FUNCTION_BLOCK fb_gm_removeLens
VAR_INPUT
	in_flg_run: BOOL;
END_VAR
VAR_OUTPUT
	out_flg_Done: BOOL;
END_VAR
VAR
	SFCInit: BOOL;
	trn_checkVacDone: BOOL;
	trn_rmoveLensThetaDone: BOOL;
	var_process: INT;
	trn_removeLensDone: BOOL;
	trn_removeLen_stocker_eject_Done : BOOL;
	trn_removeLen_stocker_fiber_Done : BOOL;
	trn_removeLen_measurement_eject_Done : BOOL;
	trn_removeLen_measurement_fiber_Done : BOOL;
	timer: TON;
	timer2: TON;
END_VAR

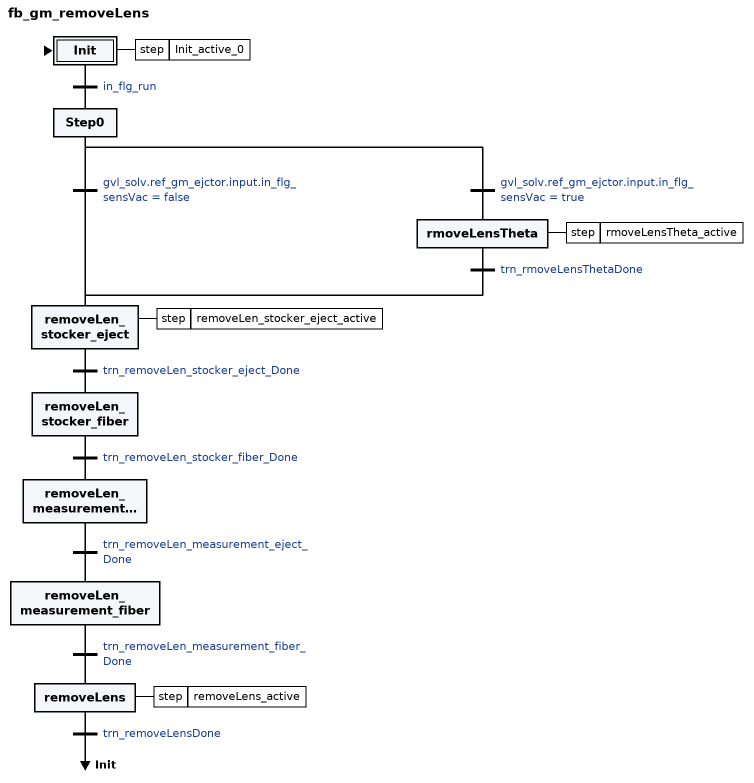
INITIAL_STEP Init:
    Init_active_0(N);  // step action
END_STEP
TRANSITION FROM Init TO Step0
    := in_flg_run;
END_TRANSITION
STEP Step0:
END_STEP
TRANSITION FROM Step0 TO removeLen_stocker_eject
    := gvl_solv.ref_gm_ejctor.input.in_flg_sensVac = false;
END_TRANSITION
TRANSITION FROM Step0 TO rmoveLensTheta
    := gvl_solv.ref_gm_ejctor.input.in_flg_sensVac = true;
END_TRANSITION
STEP rmoveLensTheta:
    rmoveLensTheta_active(N);  // step action
END_STEP
TRANSITION FROM rmoveLensTheta TO removeLen_stocker_eject
    := trn_rmoveLensThetaDone;
END_TRANSITION
STEP removeLen_stocker_eject:
    removeLen_stocker_eject_active(N);  // step action
END_STEP
TRANSITION FROM removeLen_stocker_eject TO removeLen_stocker_fiber
    := trn_removeLen_stocker_eject_Done;
END_TRANSITION
STEP removeLen_stocker_fiber:
END_STEP
TRANSITION FROM removeLen_stocker_fiber TO removeLen_measurement_eject
    := trn_removeLen_stocker_fiber_Done;
END_TRANSITION
STEP removeLen_measurement_eject:
END_STEP
TRANSITION FROM removeLen_measurement_eject TO removeLen_measurement_fiber
    := trn_removeLen_measurement_eject_Done;
END_TRANSITION
STEP removeLen_measurement_fiber:
END_STEP
TRANSITION FROM removeLen_measurement_fiber TO removeLens
    := trn_removeLen_measurement_fiber_Done;
END_TRANSITION
STEP removeLens:
    removeLens_active(N);  // step action
END_STEP
TRANSITION FROM removeLens TO Init
    := trn_removeLensDone;
END_TRANSITION

ACTION Init_active:
trn_removeLensDOne := false;
END_ACTION

ACTION Init_active_0:
out_flg_done := false;
END_ACTION

PROPERTY p_Init : BOOL
GET
p_Init := THIS^.SFCInit;
END_GET
SET
THIS^.SFCInit := p_Init;
END_SET
END_PROPERTY

ACTION removeLen_stocker_eject_active:
IF removeLen_stocker_eject._x AND removeLen_stocker_eject.x = FALSE THEN
	trn_removeLensDone := FALSE;
	timer.IN := FALSE;
	timer2.IN := FALSE;
	gvl_elecylinder.fbi_gm_axisPickUp.in_flg_run := FALSE;
	gvl_elecylinder.fbi_gm_axisPickUp.in_var_moveMode := eP_eleMoveMode.eleB;
	gvl_solv.fbi_gm_ejector.in_flg_run := FALSE;
	gvl_solv.fbi_gm_ejector.in_var_vacMode := eP_ejeVacMode.halt;
	gvl_axis.ref_r.Execute := FALSE;
	gvl_solv.fbi_gm_chuck.in_var_moveMode := eP_svMoveMode.svB;
	gvl_solv.fbi_gm_chuck.in_flg_run := FALSE;
	gvl_solv.fbi_gm_push.in_var_moveMode := eP_svMoveMode.svB;
	gvl_solv.fbi_gm_push.in_flg_run := FALSE;
	gvl_axis.ref_r.Position := gvl_param.var_productInfo[gvl_param.var_currentProductID].teachPos.gm_rotary.pickUp;
	var_process := 0;
ELSIF removeLen_stocker_eject._x AND removeLen_stocker_eject.x THEN
	CASE var_process OF
		0:
			IF gvl_io.flg_gm_fiberSens THEN
				var_process := 1;
			ELSE
				var_process := 100;
			END_IF
		1:
			
			
		
		
		100:
			trn_removeLensDone := TRUE;

	END_CASE
END_IF
END_ACTION

ACTION removeLens_active:
IF removeLens._x AND removeLens.x = FALSE THEN
	trn_removeLensDone := FALSE;
	timer.IN := FALSE;
	timer2.IN := FALSE;
	gvl_elecylinder.fbi_gm_axisPickUp.in_flg_run := FALSE;
	gvl_elecylinder.fbi_gm_axisPickUp.in_var_moveMode := eP_eleMoveMode.eleB;
	gvl_solv.fbi_gm_ejector.in_flg_run := FALSE;
	gvl_solv.fbi_gm_ejector.in_var_vacMode := eP_ejeVacMode.halt;
	gvl_axis.ref_r.Execute := FALSE;
	gvl_solv.fbi_gm_chuck.in_var_moveMode := eP_svMoveMode.svB;
	gvl_solv.fbi_gm_chuck.in_flg_run := FALSE;
	gvl_solv.fbi_gm_push.in_var_moveMode := eP_svMoveMode.svB;
	gvl_solv.fbi_gm_push.in_flg_run := FALSE;
	gvl_axis.ref_r.Position := gvl_param.var_productInfo[gvl_param.var_currentProductID].teachPos.gm_rotary.pickUp;
	var_process := 0;
ELSIF removeLens._x AND removeLens.x THEN
	CASE var_process OF
		0:
			IF gvl_io.flg_gm_fiberSens THEN
				//gvl_solv.fbi_gm_chuck.in_flg_run := TRUE;
				gvl_solv.fbi_gm_ejector.in_var_vacMode := eP_ejeVacMode.break;
				gvl_solv.fbi_gm_ejector.in_flg_run := TRUE;
				var_process := 15;
			ELSE
				gvl_solv.fbi_gm_ejector.in_var_vacMode := eP_ejeVacMode.break;
				gvl_solv.fbi_gm_ejector.in_flg_run := TRUE;
				var_process := 15;
			END_IF
		1:
			IF gvl_solv.fbi_gm_chuck.out_flg_Done THEN
				gvl_solv.fbi_gm_chuck.in_var_moveMode := eP_svMoveMode.svA;
				gvl_solv.fbi_gm_chuck.in_flg_run := FALSE;
				gvl_solv.fbi_gm_push.in_flg_run := TRUE;
				var_process := 2;
			END_IF
		2:
			IF gvl_solv.fbi_gm_push.out_flg_Done THEN
				gvl_solv.fbi_gm_push.in_var_moveMode := eP_svMoveMode.svA;
				gvl_solv.fbi_gm_push.in_flg_run := FALSE;
				var_process := 3;
			END_IF	
		3:
			gvl_axis.ref_r.Execute := TRUE;
			var_process := 4;
		4:
			IF gvl_axis.ref_r.Done THEN
				gvl_axis.ref_r.Execute := FALSE;
				var_process := 5;
			END_IF
		5:	
			gvl_solv.fbi_gm_ejector.in_flg_run := TRUE;
			gvl_elecylinder.fbi_gm_axisPickUp.in_flg_run := TRUE;
			var_process := 6;
		6:
			IF gvl_elecylinder.fbi_gm_axisPickUp.out_flg_Done THEN
				timer.IN := TRUE;
				gvl_elecylinder.fbi_gm_axisPickUp.in_flg_run := FALSE;
				var_process := 7;
			END_IF
		7:
			IF 	timer.Q THEN
				gvl_elecylinder.fbi_gm_axisPickUp.in_var_moveMode := eP_eleMoveMode.eleA;
				gvl_elecylinder.fbi_gm_axisPickUp.in_flg_run := FALSE;
				var_process := 8;
			END_IF
		8:
			gvl_solv.fbi_gm_chuck.in_flg_run := TRUE;
			gvl_solv.fbi_gm_push.in_flg_run := TRUE;
			var_process := 9;
		9:
			timer2.IN := TRUE;
			IF timer2.Q THEN
				var_process := 10;
			END_IF
			
		10:
			gvl_elecylinder.fbi_gm_axisPickUp.in_flg_run := TRUE;
			gvl_axis.ref_r.Position := gvl_param.var_productInfo[gvl_param.var_currentProductID].teachPos.gm_rotary.remove;
			var_process := 11;
		11:
			IF gvl_elecylinder.fbi_gm_axisPickUp.out_flg_Done THEN
				gvl_axis.ref_r.Execute := TRUE;
				gvl_solv.fbi_gm_ejector.in_flg_run := FALSE;
				gvl_solv.fbi_gm_ejector.in_var_vacMode := eP_ejeVacMode.break;
				var_process := 12;
			END_IF
		12:
			IF gvl_axis.ref_r.Done THEN
				gvl_axis.ref_r.Execute := FALSE;
				gvl_solv.fbi_gm_ejector.in_flg_run := TRUE;
				var_process := 13;
			END_IF
		13:
			IF gvl_solv.fbi_gm_ejector.out_flg_Done THEN
				gvl_axis.ref_r.Position := gvl_param.var_productInfo[gvl_param.var_currentProductID].teachPos.gm_rotary.origin;
				gvl_axis.ref_r.Execute := TRUE;
				var_process := 14;
			END_IF
		14:
			IF gvl_axis.ref_r.Done THEN
				gvl_axis.ref_r.Execute := FALSE;
				var_process := 15;
			END_IF
		15:
			gvl_solv.fbi_gm_ejector.in_flg_run := FALSE;
			out_flg_Done := TRUE;
			trn_removeLensDone := TRUE;
			
			
			
	END_CASE
timer(IN:= , PT:=T#0.5S , Q=> , ET=> );
timer2(IN:= , PT:=T#0.2S , Q=> , ET=> );
END_IF
END_ACTION

ACTION rmoveLensTheta_active:
IF rmoveLensTheta._x AND rmoveLensTheta.x = FALSE THEN
	var_process := 0;
	trn_rmoveLensThetaDone := FALSE;
	gvl_axis.ref_r.Execute := FALSE;
	gvl_solv.fbi_gm_ejector.in_flg_run := FALSE;
	gvl_solv.fbi_gm_ejector.in_var_vacMode := eP_ejeVacMode.break;
	gvl_axis.ref_r.Position := gvl_param.var_productInfo[gvl_param.var_currentProductID].teachPos.gm_rotary.remove;
ELSIF rmoveLensTheta._x AND rmoveLensTheta.x THEN
	CASE var_process OF
		0:
			gvl_axis.ref_r.Execute := TRUE;
			var_process := 1;
		1:
			IF gvl_axis.ref_r.Done THEN
				gvl_solv.fbi_gm_ejector.in_flg_run := TRUE;
				var_process := 2;
			END_IF
		2:
			IF gvl_solv.fbi_gm_ejector.out_flg_Done THEN
				var_process := 3;
			END_IF
		3:	
			gvl_axis.ref_r.Position := gvl_param.var_productInfo[gvl_param.var_currentProductID].teachPos.gm_rotary.pickUp;
			gvl_axis.ref_r.Execute := FALSE;
			var_process := 4;
		4:
			gvl_axis.ref_r.Execute := TRUE;
			var_process := 5;
		5:
			IF gvl_axis.ref_r.Done THEN
				trn_rmoveLensThetaDone := TRUE;
			END_IF
	END_CASE
END_IF
END_ACTION

END_FUNCTION_BLOCK

(* stored: Version 1.1.0.1, ProductVersion 3.1.4024.12
   POU fb_gm_removeLens: Id {a652fa65-7059-4187-8597-894c14dd1d48}, SpecialFunc None
   Action Init_active: Id {89c4f83a-a694-4f99-ab4b-138e7e567033}
   Action Init_active_0: Id {a0514581-c5e7-491a-b4b1-406e48d7cff9}
   Property p_Init: Id {ed900328-9a15-4edc-b486-c4dfbede0b7f}
   Get Get: Id {5f4c62d5-a4e7-4781-a31e-30e17f86c1cb}
   Set Set: Id {0f71ef2c-6bc4-448b-9e0a-6dc10fb66dbd}
   Action removeLen_stocker_eject_active: Id {557eafa1-9040-433e-a5c7-b763c076be3f}
   Action removeLens_active: Id {1ea01717-d15e-4817-bcea-abd2ac008929}
   Action rmoveLensTheta_active: Id {5b3b94fd-3952-4c3f-998a-e4be43ed7eea} *)
